// TIA Portal V18 export
FUNCTION_BLOCK "valve"   // FB8, LAD
{ S7_Optimized_Access := 'FALSE' }
VERSION : 0.1
// stored: AutoNumber true, IsIECCheckEnabled false, SetENOAutomatically false, UDAEnableTagReadback false
   VAR_INPUT
      "A/M" : Bool;
      open_auto : Bool;
      open_man : Bool;
      fbk_open : Bool;
      fbk_close : Bool;
      reset : Bool;
      intl : Bool;
      Mon_En : Bool;
      mon_sp : Time;
      run_fb : Bool;
      stop_fb : Bool;
   END_VAR
   VAR_OUTPUT
      "open/close" : Bool;
      fault : Bool;
      status : Int;
   END_VAR
   VAR DB_SPECIFIC
      open_fault : Bool;
      close_fault : Bool;
      IEC_Timer_0_Instance { S7_SetPoint := 'True'} : TON_TIME;
      IEC_Timer_0_Instance_1 { S7_SetPoint := 'True'} : TON_TIME;
      mon : Int;
      pulse : Bool;
      pulse1 : Bool;
      mon1 : Int;
      IEC_Timer_0_Instance_2 { S7_SetPoint := 'True'} : TON_TIME;
   END_VAR
   VAR_TEMP   // added for the SCL form of the ladder/FBD networks
      _w1 : Bool;
   END_VAR
BEGIN

REGION Network 1
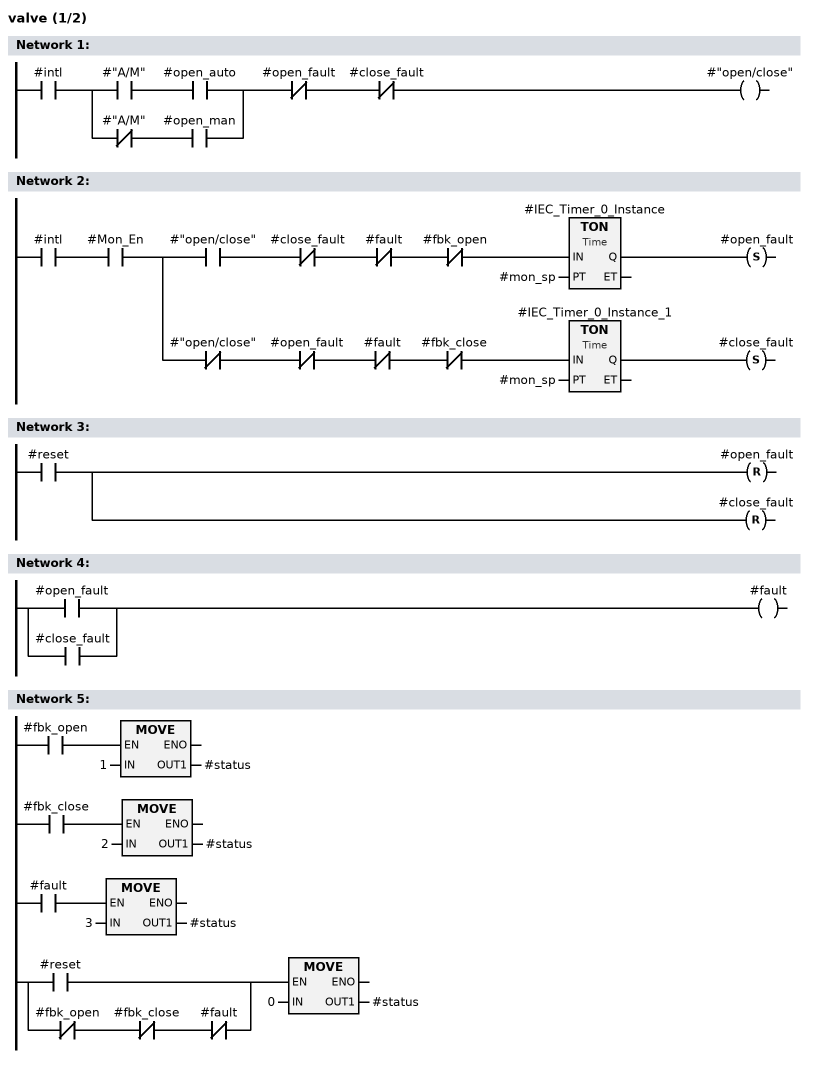
   RUNG wire#powerrail
      Contact( #intl )
      wire#w1
      Contact( #"A/M" )
      Contact( #open_auto )
      wire#w2
      I_Contact( #open_fault )
      I_Contact( #close_fault )
      Coil( #"open/close" )
   END_RUNG
   RUNG wire#w1
      I_Contact( #"A/M" )
      Contact( #open_man )
   END_RUNG wire#w2
   // the same network as SCL:
   #"open/close" := #intl AND ((#"A/M" AND #open_auto) OR (NOT #"A/M" AND #open_man)) AND NOT #open_fault AND NOT #close_fault;
END_REGION

REGION Network 2
   RUNG wire#powerrail
      Contact( #intl )
      Contact( #Mon_En )
      wire#w1
      Contact( #"open/close" )
      I_Contact( #close_fault )
      I_Contact( #fault )
      I_Contact( #fbk_open )
      { S7_Templates := "time_type := Time" } #IEC_Timer_0_Instance.TON(pt := #mon_sp, et =>)
      S_Coil( #open_fault )
   END_RUNG
   RUNG wire#w1
      I_Contact( #"open/close" )
      I_Contact( #open_fault )
      I_Contact( #fault )
      I_Contact( #fbk_close )
      { S7_Templates := "time_type := Time" } #IEC_Timer_0_Instance_1.TON(pt := #mon_sp, et =>)
      S_Coil( #close_fault )
   END_RUNG
   // the same network as SCL:
   #_w1 := #intl AND #Mon_En;
   #IEC_Timer_0_Instance(IN := #_w1 AND #"open/close" AND NOT #close_fault AND NOT #fault AND NOT #fbk_open,   // TON
                         PT := #mon_sp);
   IF #IEC_Timer_0_Instance.Q THEN #open_fault := TRUE; END_IF;
   #IEC_Timer_0_Instance_1(IN := #_w1 AND NOT #"open/close" AND NOT #open_fault AND NOT #fault AND NOT #fbk_close,   // TON
                           PT := #mon_sp);
   IF #IEC_Timer_0_Instance_1.Q THEN #close_fault := TRUE; END_IF;
END_REGION

REGION Network 3
   RUNG wire#powerrail
      Contact( #reset )
      wire#w1
      R_Coil( #open_fault )
   END_RUNG
   RUNG wire#w1
      R_Coil( #close_fault )
   END_RUNG
   // the same network as SCL:
   IF #reset THEN
       #open_fault := FALSE;
       #close_fault := FALSE;
   END_IF;
END_REGION

REGION Network 4
   RUNG wire#powerrail
      Contact( #open_fault )
      wire#w1
      Coil( #fault )
   END_RUNG
   RUNG wire#powerrail
      Contact( #close_fault )
   END_RUNG wire#w1
   // the same network as SCL:
   #fault := #open_fault OR #close_fault;
END_REGION

REGION Network 5
   RUNG wire#powerrail
      Contact( #fbk_open )
      Move(in := 1, out1 => #status)
   END_RUNG
   RUNG wire#powerrail
      Contact( #fbk_close )
      Move(in := 2, out1 => #status)
   END_RUNG
   RUNG wire#powerrail
      Contact( #fault )
      Move(in := 3, out1 => #status)
   END_RUNG
   RUNG wire#powerrail
      Contact( #reset )
      wire#w1
      Move(in := 0, out1 => #status)
   END_RUNG
   RUNG wire#powerrail
      I_Contact( #fbk_open )
      I_Contact( #fbk_close )
      I_Contact( #fault )
   END_RUNG wire#w1
   // the same network as SCL:
   IF #fbk_open THEN #status := 1; END_IF;
   IF #fbk_close THEN #status := 2; END_IF;
   IF #fault THEN #status := 3; END_IF;
   IF #reset OR (NOT #fbk_open AND NOT #fbk_close AND NOT #fault) THEN #status := 0; END_IF;
END_REGION

REGION Network 7
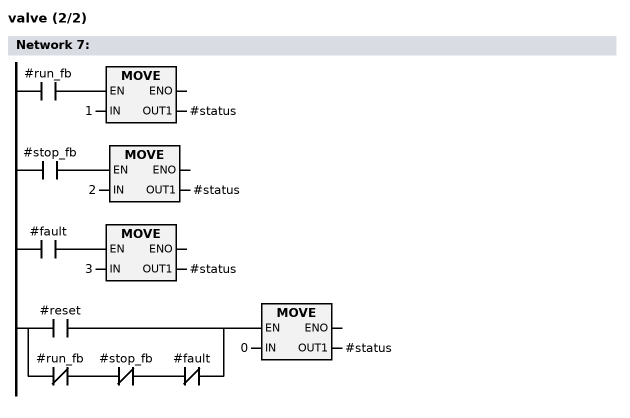
   RUNG wire#powerrail
      Contact( #run_fb )
      Move(in := 1, out1 => #status)
   END_RUNG
   RUNG wire#powerrail
      Contact( #stop_fb )
      Move(in := 2, out1 => #status)
   END_RUNG
   RUNG wire#powerrail
      Contact( #fault )
      Move(in := 3, out1 => #status)
   END_RUNG
   RUNG wire#powerrail
      Contact( #reset )
      wire#w1
      Move(in := 0, out1 => #status)
   END_RUNG
   RUNG wire#powerrail
      I_Contact( #run_fb )
      I_Contact( #stop_fb )
      I_Contact( #fault )
   END_RUNG wire#w1
   // the same network as SCL:
   IF #run_fb THEN #status := 1; END_IF;
   IF #stop_fb THEN #status := 2; END_IF;
   IF #fault THEN #status := 3; END_IF;
   IF #reset OR (NOT #run_fb AND NOT #stop_fb AND NOT #fault) THEN #status := 0; END_IF;
END_REGION
END_FUNCTION_BLOCK
